Staubli VAL3: delJRsArray.pgx

public program delJRsArray(jointRs& x_In[], num x_nNum)
  local num l_nSize
begin
  //删除字符串数组
  //x_sStrIn:返回的新数组
  //x_nNum:删除数组个数
  //取整
  x_nNum=roundDown(x_nNum)
  //
  l_nSize=size(x_In)
  if l_nSize<=1
    return
  endIf
  //
  if x_nNum>=l_nSize
    x_nNum=l_nSize-1
  endIf
  //
  while x_nNum>=1
    delete(x_In[0])
    x_nNum=x_nNum-1
  endWhile
end
